{attribute 'enable_dynamic_creation'}
TYPE NodeINT :
STRUCT
	data : INT;
	next : POINTER TO NodeINT;
END_STRUCT
END_TYPE

(* stored: Version 1.1.0.1, ProductVersion 3.1.4024.11
   DUT NodeINT: Id {ec13c4f1-266e-482d-9b20-9541e4253173} *)
